INTERFACE I_Cylinder

PROPERTY bState_AtBasePos : BOOL
GET
END_GET
END_PROPERTY

PROPERTY bState_AtWorkPos : BOOL
GET
END_GET
END_PROPERTY

PROPERTY bState_MoveToWork : BOOL
GET
END_GET
END_PROPERTY

METHOD MoveToBase
VAR_INPUT
END_VAR
END_METHOD

METHOD MoveToWork
VAR_INPUT
END_VAR
END_METHOD

METHOD Reset
VAR_INPUT
END_VAR
END_METHOD

END_INTERFACE

(* stored: Version 1.1.0.1, ProductVersion 3.1.4024.2
   Itf I_Cylinder: Id {999197fd-9016-43c5-9286-554445a30fcc}
   Property bState_AtBasePos: Id {870102fa-bd15-471e-89f6-7f98c7c6a1e1}
   Get Get: Id {5f03cda0-73ef-4332-a87e-0bad6e137d09}
   Property bState_AtWorkPos: Id {196503f9-7fb0-4e10-b1c6-6ec1d5f973a3}
   Get Get: Id {696b45f5-b3b7-4502-b54f-0ce90e0b7895}
   Property bState_MoveToWork: Id {b936c052-6de0-49d1-8917-7b0b5644a0f9}
   Get Get: Id {b6ea64c0-3021-4c67-9ff9-6567ec946641}
   Method MoveToBase: Id {743e8bca-f87c-47dc-b63d-c43eea822e03}
   Method MoveToWork: Id {d78a2c2e-cf00-47dd-a32e-dbbdb7165b31}
   Method Reset: Id {9f27252d-8587-4a98-b79c-05aaf0568907} *)
